(* PLC project AKS_v2.project, Prosoft-Systems Ltd. Astra.IDE Astra.IDE_V1.7.2.1 *)
(* stored: creationDateTime 2025-07-24T10:35:59.4336606, modificationDateTime 2025-07-24T08:15:04.4598718 *)

{attribute 'object_name' := 'AI__1'}
PROGRAM AI__1_1
  VAR
    DI_DI : FB_DI;
    A : BOOL;
    B : BOOL;
  END_VAR

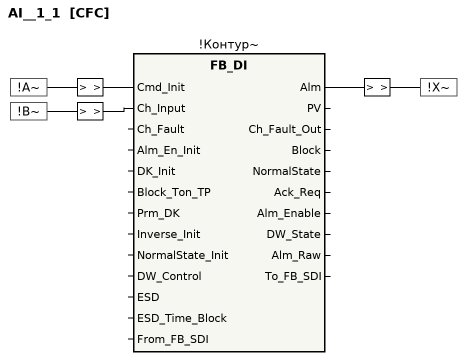
(* CFC diagram, written out as Structured Text *)
!X~ := !Контур~.Alm;
!Контур~(Cmd_Init := !A~, Ch_Input := !B~);
END_PROGRAM
